FUNCTION_BLOCK FB_Methods
VAR
	count : LREAL;
END_VAR

{attribute 'TcRpcEnable'}
{attribute 'OPC.UA.DA.Description' := 'Returns array of INT'}
METHOD M_Array_1 : ARRAY[0..2] OF INT
VAR_INPUT
END_VAR
VAR
	aTest : ARRAY[0..2] OF INT;
END_VAR
aTest[0] := 1;
aTest[1] := 2;
aTest[2] := 3;
M_Array_1 := aTest;
END_METHOD

{attribute 'TcRpcEnable'}
{attribute 'OPC.UA.DA.Description' := 'Returns array of INT'}
METHOD M_Array_2 : ARRAY[0..9] OF INT
VAR_INPUT
	aTest : ARRAY[0..9] OF INT;
END_VAR
M_Array_2 := aTest;
END_METHOD

{attribute 'TcRpcEnable'}
{attribute 'OPC.UA.DA.Description' := 'Returns simple complex type'}
METHOD M_Complex_1 : ST_Complex_1
count :=count+1;
M_Complex_1.a := 1;
M_Complex_1.b := 2;
END_METHOD

{attribute 'TcRpcEnable'}
{attribute 'OPC.UA.DA.Description' := 'InOut argument is a simple complex type'}
METHOD M_Complex_2 : ST_Complex_1
VAR_INPUT
	in : ST_Complex_1;
END_VAR
count :=count+1;
M_Complex_2.a := in.a + 1;
M_Complex_2.b := in.b + 1;
END_METHOD

{attribute 'TcRpcEnable'}
{attribute 'OPC.UA.DA.Description' := 'Method without InOut arguments'}
METHOD M_NoArgs
VAR_INPUT
END_VAR
count :=count+1;
END_METHOD

END_FUNCTION_BLOCK

(* stored: Version 1.1.0.1
   POU FB_Methods: Id {daffb5d3-941c-4f0b-84c9-30e8405c541a}, SpecialFunc None
   Method M_Array_1: Id {15221446-3a21-4239-b8a3-00f4dce8483f}
   Method M_Array_2: Id {fa68f12f-e6d5-42bd-ab0a-04def1c9d2b8}
   Method M_Complex_1: Id {5806ee66-5b5d-4b39-9af1-417eb561995c}
   Method M_Complex_2: Id {4bc1313e-5501-4cb5-9aba-f48f187748a6}
   Method M_NoArgs: Id {d2f58dae-424c-4621-996c-d0582f3e8ba7} *)
